PROGRAM P_OnResetClick
VAR
END_VAR

F_AuswertungBefehlstastenVonTP(tastenWert := CVL.RESET_BUTTON);
F_ResetEndSchalterFehler();

END_PROGRAM

(* stored: Version 1.1.0.1, ProductVersion 3.1.4024.3
   POU P_OnResetClick: Id {ffc97bad-9301-49cf-89e6-7d539a19fd85}, SpecialFunc None *)
